(* IEC 61131-3 sources: eCockpitGit/test_project/src/%F%00 Library/%F%JSON/%POU%FB_JSONWriter/%F%Protected, 5 files *)

(* ---- %METH%addChar.st ---- *)
//This adds a character to the JSON buffer
// |**Version**|**Author**| **Date** |**Changes**
// | 1         | NSN      | 22-06-20 | Creation
METHOD PROTECTED addChar
VAR_INPUT
	char			:EASCII;
END_VAR
(*%!%__DELIMITER__%!%*)
IF ready THEN		//It only runs when a buffer has been initialized
	IF bufferPosition < bufferMaxADR THEN	//In normal conditions
		bufferPosition^		:=		char;
		bufferPosition		:=		bufferPosition + 1;
	ELSE									//When the last address is encountered, the end of buffer variable is set true
		bufferInvalid		:=		TRUE;
	END_IF
END_IF

(* ---- %METH%addNewLine.st ---- *)
//This adds a new line and the appropriate amount of tabs
// |**Version**|**Author**| **Date** |**Changes**
// | 1         | NSN      | 22-06-20 | Creation
METHOD PROTECTED addNewLine
VAR
	i				:WORD;
END_VAR
(*%!%__DELIMITER__%!%*)
IF ready THEN
	//New Line
	addChar(char := EASCII.LF);
	//Tabs are added
	IF treeLevel > 0 THEN
		FOR i := treeLevel TO 1 BY -1 DO
			addChar(char := EASCII.Tab);
		END_FOR
	END_IF
END_IF

(* ---- %METH%addString.st ---- *)
//This adds a string of text to the JSON buffer
//Illigal characters { , } , " they will be skipped
// |**Version**|**Author**| **Date** |**Changes**
// | 1         | NSN      | 22-06-20 | Creation
METHOD PROTECTED addString
VAR_INPUT
	pString			:POINTER TO BYTE;	//Address of string for the comment text
END_VAR
(*%!%__DELIMITER__%!%*)
IF ready THEN		//It only runs when a buffer has been initialized
	IF pString <> 0 THEN						//Checks if stringaddress is not empty
		WHILE pString^ <> EASCII.Null DO			//Runs until null is detected
			IF bufferPosition < bufferMaxADR THEN	//In normal conditions
				IF pString^ = EASCII.DoubleQoute THEN
					bufferPosition^	:=		EASCII.BackSlash;
					bufferPosition	:=		bufferPosition + 1;
				END_IF
				bufferPosition^		:=		pString^;
				pString				:=		pString + 1;
				bufferPosition		:=		bufferPosition + 1;
			ELSE								//When the last address is encountered, the end of buffer variable is set true
				bufferInvalid		:=		TRUE;
				EXIT;
			END_IF
		END_WHILE
	END_IF
END_IF

(* ---- %METH%addStringRaw.st ---- *)
//This adds a string of text to the JSON buffer
//Illigal characters { , } , " they will be skipped
// |**Version**|**Author**| **Date** |**Changes**
// | 1         | NSN      | 22-06-20 | Creation
METHOD PROTECTED addStringRaw
VAR_INPUT
	pString			:POINTER TO BYTE;	//Address of string for the comment text
END_VAR
(*%!%__DELIMITER__%!%*)
IF ready THEN		//It only runs when a buffer has been initialized
	IF pString <> 0 THEN						//Checks if stringaddress is not empty
		WHILE pString^ <> EASCII.Null DO			//Runs until null is detected
			IF bufferPosition < bufferMaxADR THEN	//In normal conditions
				bufferPosition^		:=		pString^;
				pString				:=		pString + 1;
				bufferPosition		:=		bufferPosition + 1;
			ELSE
				bufferInvalid		:=		TRUE;
				EXIT;
			END_IF
		END_WHILE
	END_IF
END_IF

(* ---- %METH%addStringRawLen.st ---- *)
//This adds a string of text to the JSON buffer
//Illigal characters { , } , " they will be skipped
// |**Version**|**Author**| **Date** |**Changes**
// | 1         | NSN      | 22-06-20 | Creation
METHOD PROTECTED addStringRawLen
VAR_INPUT
	pString			:POINTER TO EASCII;	//Address of string for the comment text
	len				:DWORD;				//Amount of bytes to write
END_VAR
(*%!%__DELIMITER__%!%*)
IF ready THEN		//It only runs when a buffer has been initialized
	IF pString <> 0 THEN								//Checks if stringaddress is not empty
		WHILE pString^ <> EASCII.Null AND len > 0 DO	//Runs until null is detected
			IF bufferPosition < bufferMaxADR THEN		//In normal conditions
				bufferPosition^		:=		pString^;
				pString				:=		pString + 1;
				bufferPosition		:=		bufferPosition + 1;
				len					:=		len - 1;
			ELSE
				bufferInvalid		:=		TRUE;
				EXIT;
			END_IF
		END_WHILE
	END_IF
END_IF
